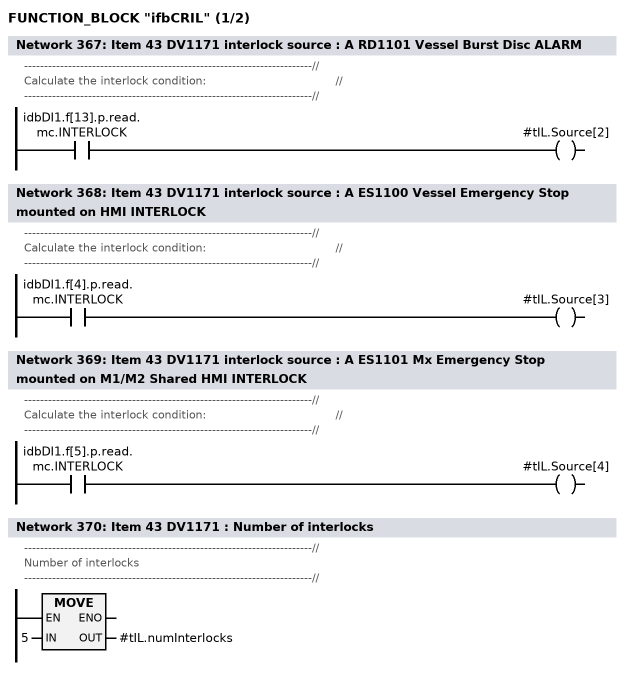
    A idbDI1.f[13].p.read.mc.INTERLOCK;
    = #tIL.Source[2];

NETWORK
TITLE = Item 43 DV1171 interlock source : A ES1100 Vessel Emergency Stop mounted on HMI INTERLOCK
    //------------------------------------------------------------------------//
    // Calculate the interlock condition:                                     //
    //------------------------------------------------------------------------//
    A idbDI1.f[4].p.read.mc.INTERLOCK;
    = #tIL.Source[3];

NETWORK
TITLE = Item 43 DV1171 interlock source : A ES1101 Mx Emergency Stop mounted on M1/M2 Shared HMI INTERLOCK
    //------------------------------------------------------------------------//
    // Calculate the interlock condition:                                     //
    //------------------------------------------------------------------------//
    A idbDI1.f[5].p.read.mc.INTERLOCK;
    = #tIL.Source[4];


NETWORK
TITLE = Item 43 DV1171 : Number of interlocks
    //------------------------------------------------------------------------//
    // Number of interlocks
    //------------------------------------------------------------------------//
    L 5;
    T #tIL.numInterlocks;

NETWORK
TITLE = Item 43 DV1171 : Aggregate individual interlocks into overall INTERLOCK flag
    //------------------------------------------------------------------------//
    // Determine if an interlock is raised:                                   //
    //------------------------------------------------------------------------//
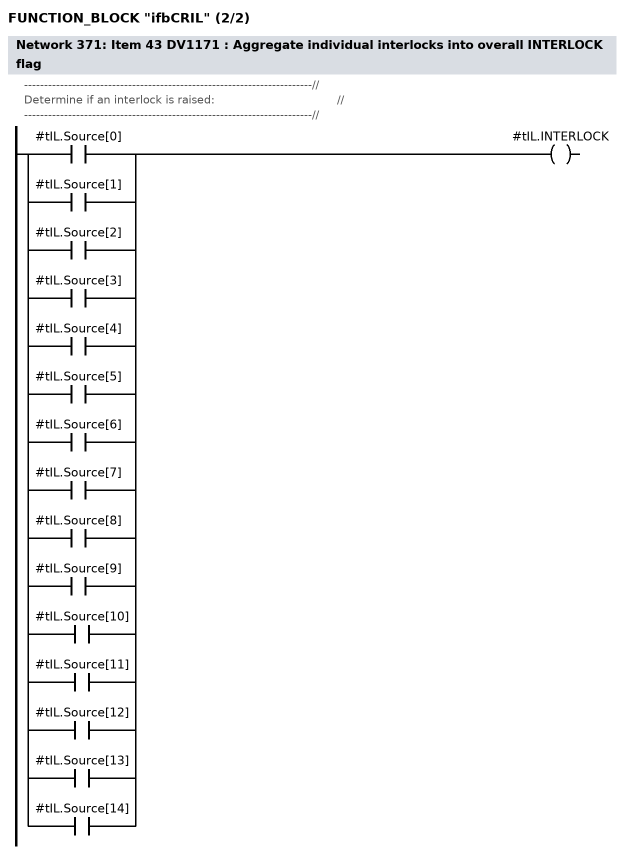
    O #tIL.Source[0];
    O #tIL.Source[1];
    O #tIL.Source[2];
    O #tIL.Source[3];
    O #tIL.Source[4];
    O #tIL.Source[5];
    O #tIL.Source[6];
    O #tIL.Source[7];
    O #tIL.Source[8];
    O #tIL.Source[9];
    O #tIL.Source[10];
    O #tIL.Source[11];
    O #tIL.Source[12];
    O #tIL.Source[13];
    O #tIL.Source[14];
    = #tIL.INTERLOCK;

NETWORK
TITLE = Item 43 DV1171 : Update the instance data
    //------------------------------------------------------------------------//
    // Update the instance DB with the calculated interlock flags:            //
    //------------------------------------------------------------------------//
    CALL MOVE
    {value_type := 'Variant'}
    (   IN                   := #tIL ,
        OUT                  := #p[43]
    );

NETWORK
TITLE = Item 44 DV1173 : MMFLx Inline Heat Exchanger inlet valve initialise variables
    //------------------------------------------------------------------------//
    // CRITICAL INTERLOCK   CRITICAL INTERLOCK   CRITICAL INTERLOCK   CRITICA //
    // CRITICAL INTERLOCK   CRITICAL INTERLOCK   CRITICAL INTERLOCK   CRITICA //
    //                                                                        //
    // Clear the interlock flag:                                              //
    //------------------------------------------------------------------------//
    A "alwaysLow";
    = #tIL.INTERLOCK;

    //------------------------------------------------------------------------//
    // Clear all interlock values to initialise them to off:                  //
    //------------------------------------------------------------------------//
    CALL FILL_BLK
    {value_type := 'Bool', count_type := 'UInt'}
    (   IN                   := 0 ,
        COUNT                := 15 ,
        OUT                  := #tIL.Source[0]
    );


NETWORK
TITLE = Item 44 DV1173 interlock source : AN ZSC1113 MMFLx Filtration Inlet Flowpath Indicator IN   AN ZSC1115 MMFLx Filtration Inlet CIP & SIP Flowpath Indicator IN
    //------------------------------------------------------------------------//
    // Calculate the interlock condition:                                     //
    //------------------------------------------------------------------------//
    AN(;
    L "idbZSC2".f[5].p.read.mc.STATE;
    L "dbCONST".BLK.ZSC2.STATE.IN;
    ==I;
    );
AN(;
    L "idbZSC2".f[6].p.read.mc.STATE;
    L "dbCONST".BLK.ZSC2.STATE.IN;
    ==I;
    );
    = #tIL.Source[0];

NETWORK
TITLE = Item 44 DV1173 interlock source : A RD1101 Vessel Burst Disc ALARM
    //------------------------------------------------------------------------//
    // Calculate the interlock condition:                                     //
    //------------------------------------------------------------------------//
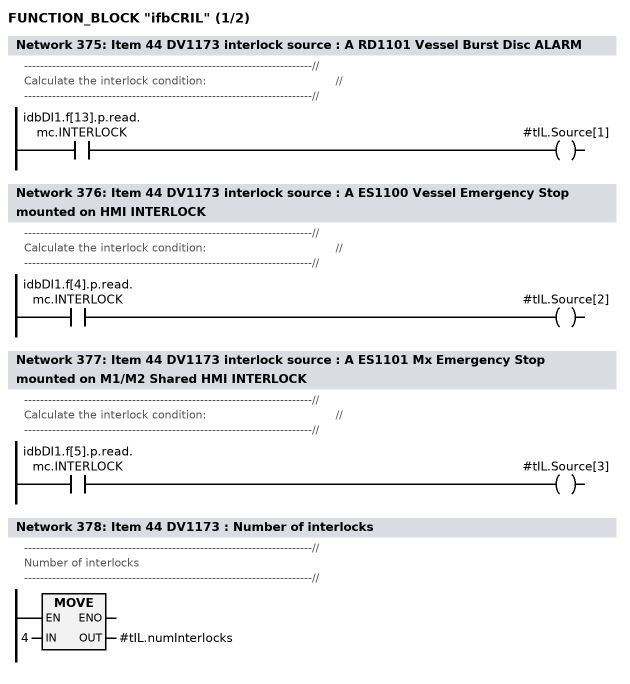
    A idbDI1.f[13].p.read.mc.INTERLOCK;
    = #tIL.Source[1];

NETWORK
TITLE = Item 44 DV1173 interlock source : A ES1100 Vessel Emergency Stop mounted on HMI INTERLOCK
    //------------------------------------------------------------------------//
    // Calculate the interlock condition:                                     //
    //------------------------------------------------------------------------//
    A idbDI1.f[4].p.read.mc.INTERLOCK;
    = #tIL.Source[2];

NETWORK
TITLE = Item 44 DV1173 interlock source : A ES1101 Mx Emergency Stop mounted on M1/M2 Shared HMI INTERLOCK
    //------------------------------------------------------------------------//
    // Calculate the interlock condition:                                     //
    //------------------------------------------------------------------------//
    A idbDI1.f[5].p.read.mc.INTERLOCK;
    = #tIL.Source[3];


NETWORK
TITLE = Item 44 DV1173 : Number of interlocks
    //------------------------------------------------------------------------//
    // Number of interlocks
    //------------------------------------------------------------------------//
    L 4;
    T #tIL.numInterlocks;

NETWORK
TITLE = Item 44 DV1173 : Aggregate individual interlocks into overall INTERLOCK flag
    //------------------------------------------------------------------------//
    // Determine if an interlock is raised:                                   //
    //------------------------------------------------------------------------//
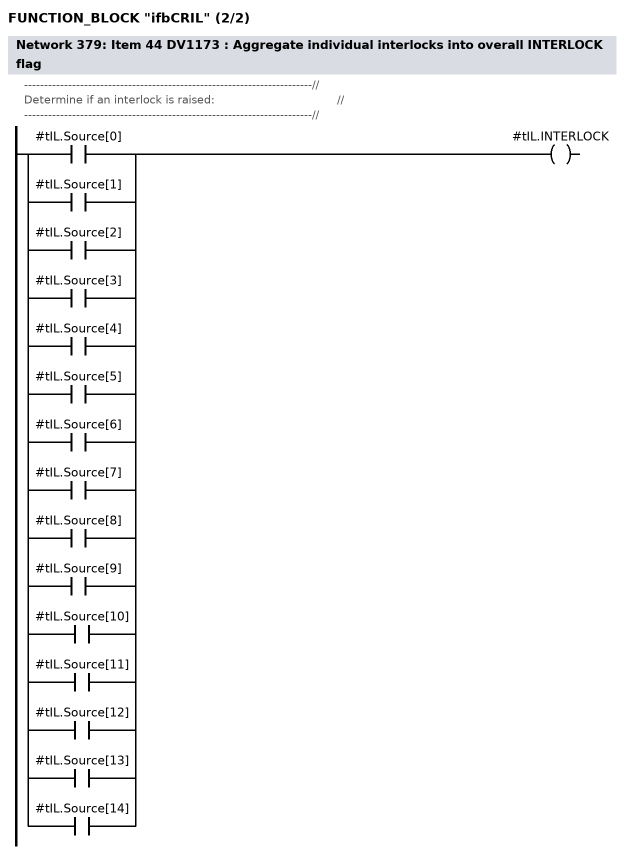
    O #tIL.Source[0];
    O #tIL.Source[1];
    O #tIL.Source[2];
    O #tIL.Source[3];
    O #tIL.Source[4];
    O #tIL.Source[5];
    O #tIL.Source[6];
    O #tIL.Source[7];
    O #tIL.Source[8];
    O #tIL.Source[9];
    O #tIL.Source[10];
    O #tIL.Source[11];
    O #tIL.Source[12];
    O #tIL.Source[13];
    O #tIL.Source[14];
    = #tIL.INTERLOCK;

NETWORK
TITLE = Item 44 DV1173 : Update the instance data
    //------------------------------------------------------------------------//
    // Update the instance DB with the calculated interlock flags:            //
    //------------------------------------------------------------------------//
    CALL MOVE
    {value_type := 'Variant'}
    (   IN                   := #tIL ,
        OUT                  := #p[44]
    );

NETWORK
TITLE = Item 45 DV2101 : Vent Valve initialise variables
    //------------------------------------------------------------------------//
    // CRITICAL INTERLOCK   CRITICAL INTERLOCK   CRITICAL INTERLOCK   CRITICA //
    // CRITICAL INTERLOCK   CRITICAL INTERLOCK   CRITICAL INTERLOCK   CRITICA //
    //                                                                        //
    // Clear the interlock flag:                                              //
    //------------------------------------------------------------------------//
    A "alwaysLow";
    = #tIL.INTERLOCK;

    //------------------------------------------------------------------------//
    // Clear all interlock values to initialise them to off:                  //
    //------------------------------------------------------------------------//
    CALL FILL_BLK
    {value_type := 'Bool', count_type := 'UInt'}
    (   IN                   := 0 ,
        COUNT                := 15 ,
        OUT                  := #tIL.Source[0]
    );


NETWORK
TITLE = Item 45 DV2101 interlock source : A RD2101 Vessel Burst Disc ALARM
    //------------------------------------------------------------------------//
    // Calculate the interlock condition:                                     //
    //------------------------------------------------------------------------//
    A idbDI1.f[14].p.read.mc.INTERLOCK;
    = #tIL.Source[0];

NETWORK
TITLE = Item 45 DV2101 interlock source : A ES2100 Vessel Emergency Stop mounted on HMI INTERLOCK
    //------------------------------------------------------------------------//
    // Calculate the interlock condition:                                     //
    //------------------------------------------------------------------------//
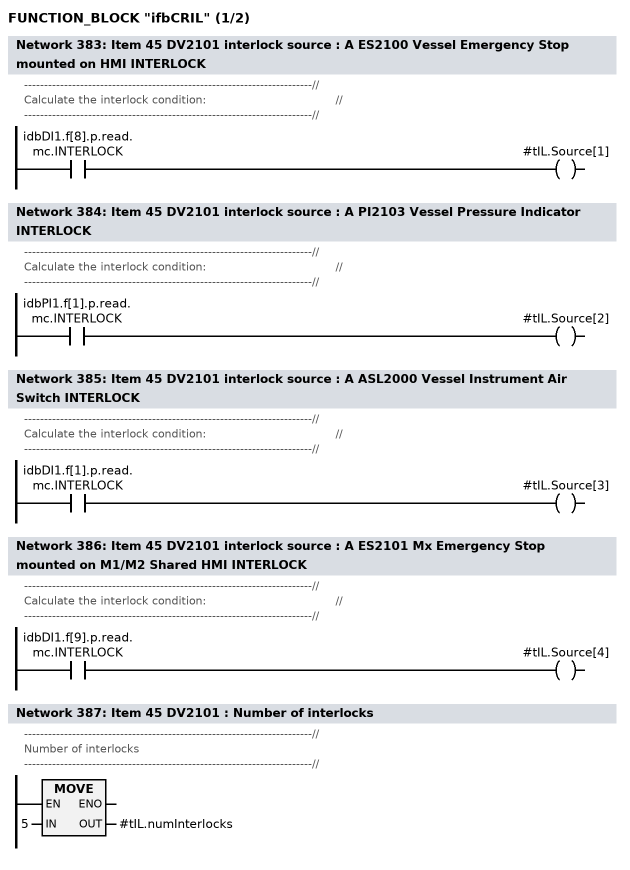
    A idbDI1.f[8].p.read.mc.INTERLOCK;
    = #tIL.Source[1];

NETWORK
TITLE = Item 45 DV2101 interlock source : A PI2103 Vessel Pressure Indicator INTERLOCK
    //------------------------------------------------------------------------//
    // Calculate the interlock condition:                                     //
    //------------------------------------------------------------------------//
    A idbPI1.f[1].p.read.mc.INTERLOCK;
    = #tIL.Source[2];

NETWORK
TITLE = Item 45 DV2101 interlock source : A ASL2000 Vessel Instrument Air Switch INTERLOCK
    //------------------------------------------------------------------------//
    // Calculate the interlock condition:                                     //
    //------------------------------------------------------------------------//
    A idbDI1.f[1].p.read.mc.INTERLOCK;
    = #tIL.Source[3];

NETWORK
TITLE = Item 45 DV2101 interlock source : A ES2101 Mx Emergency Stop mounted on M1/M2 Shared HMI INTERLOCK
    //------------------------------------------------------------------------//
    // Calculate the interlock condition:                                     //
    //------------------------------------------------------------------------//
    A idbDI1.f[9].p.read.mc.INTERLOCK;
    = #tIL.Source[4];


NETWORK
TITLE = Item 45 DV2101 : Number of interlocks
    //------------------------------------------------------------------------//
    // Number of interlocks
    //------------------------------------------------------------------------//
    L 5;
    T #tIL.numInterlocks;

NETWORK
TITLE = Item 45 DV2101 : Aggregate individual interlocks into overall INTERLOCK flag
    //------------------------------------------------------------------------//
    // Determine if an interlock is raised:                                   //
    //------------------------------------------------------------------------//
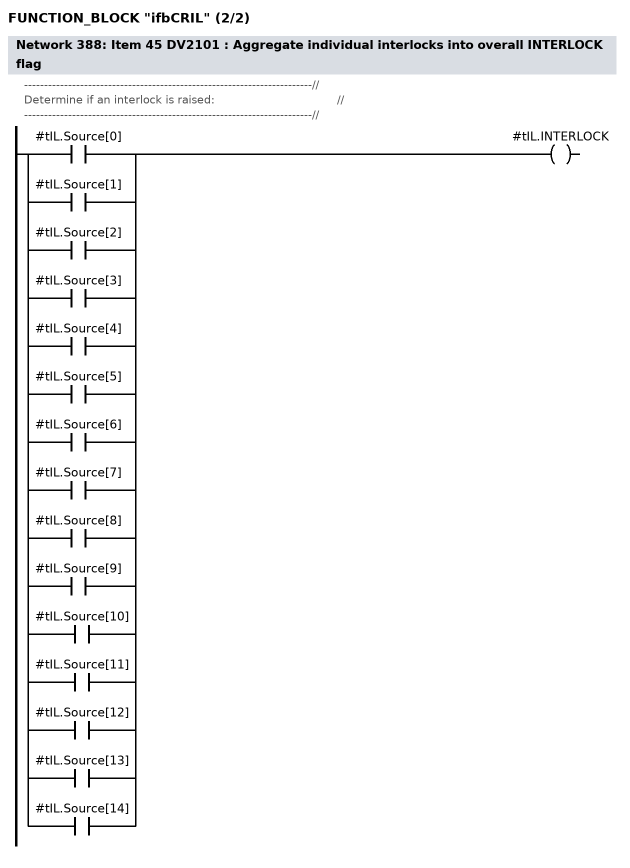
    O #tIL.Source[0];
    O #tIL.Source[1];
    O #tIL.Source[2];
    O #tIL.Source[3];
    O #tIL.Source[4];
    O #tIL.Source[5];
    O #tIL.Source[6];
    O #tIL.Source[7];
    O #tIL.Source[8];
    O #tIL.Source[9];
    O #tIL.Source[10];
    O #tIL.Source[11];
    O #tIL.Source[12];
    O #tIL.Source[13];
    O #tIL.Source[14];
    = #tIL.INTERLOCK;

NETWORK
TITLE = Item 45 DV2101 : Update the instance data
    //------------------------------------------------------------------------//
    // Update the instance DB with the calculated interlock flags:            //
    //------------------------------------------------------------------------//
    CALL MOVE
    {value_type := 'Variant'}
    (   IN                   := #tIL ,
        OUT                  := #p[45]
    );

NETWORK
TITLE = Item 46 DV2103 : HP CA Supply Valve initialise variables
    //------------------------------------------------------------------------//
    // CRITICAL INTERLOCK   CRITICAL INTERLOCK   CRITICAL INTERLOCK   CRITICA //
    // CRITICAL INTERLOCK   CRITICAL INTERLOCK   CRITICAL INTERLOCK   CRITICA //
    //                                                                        //
    // Clear the interlock flag:                                              //
    //------------------------------------------------------------------------//
    A "alwaysLow";
    = #tIL.INTERLOCK;

    //------------------------------------------------------------------------//
    // Clear all interlock values to initialise them to off:                  //
    //------------------------------------------------------------------------//
    CALL FILL_BLK
    {value_type := 'Bool', count_type := 'UInt'}
    (   IN                   := 0 ,
        COUNT                := 15 ,
        OUT                  := #tIL.Source[0]
    );


NETWORK
TITLE = Item 46 DV2103 interlock source : A RD2101 Vessel Burst Disc ALARM
    //------------------------------------------------------------------------//
    // Calculate the interlock condition:                                     //
    //------------------------------------------------------------------------//
    A idbDI1.f[14].p.read.mc.INTERLOCK;
    = #tIL.Source[0];

NETWORK
TITLE = Item 46 DV2103 interlock source : A ES2100 Vessel Emergency Stop mounted on HMI INTERLOCK
    //------------------------------------------------------------------------//
    // Calculate the interlock condition:                                     //
    //------------------------------------------------------------------------//
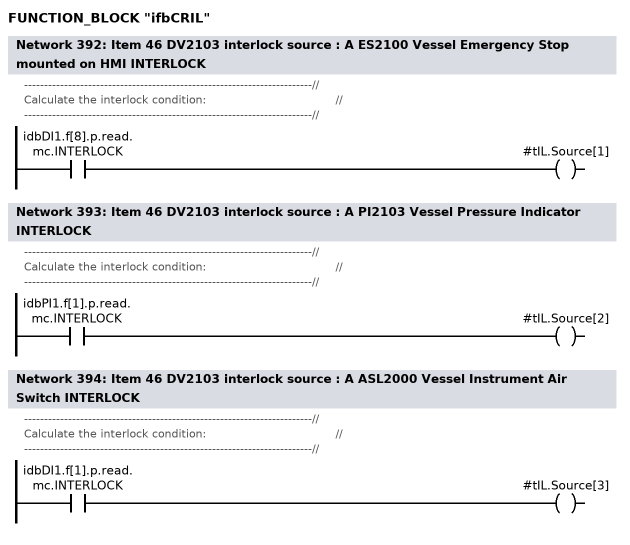
    A idbDI1.f[8].p.read.mc.INTERLOCK;
    = #tIL.Source[1];

NETWORK
TITLE = Item 46 DV2103 interlock source : A PI2103 Vessel Pressure Indicator INTERLOCK
    //------------------------------------------------------------------------//
    // Calculate the interlock condition:                                     //
    //------------------------------------------------------------------------//
    A idbPI1.f[1].p.read.mc.INTERLOCK;
    = #tIL.Source[2];

NETWORK
TITLE = Item 46 DV2103 interlock source : A ASL2000 Vessel Instrument Air Switch INTERLOCK
    //------------------------------------------------------------------------//
    // Calculate the interlock condition:                                     //
    //------------------------------------------------------------------------//
    A idbDI1.f[1].p.read.mc.INTERLOCK;
    = #tIL.Source[3];

NETWORK
TITLE = Item 46 DV2103 interlock source : AN ZSC2101 Vessel Manway Closed Indicator CLOSED
    //------------------------------------------------------------------------//
    // Calculate the interlock condition:                                     //
    //------------------------------------------------------------------------//
    AN(;
    L "idbZSC1".f[1].p.read.mc.STATE;
    L "dbCONST".BLK.ZSC1.STATE.CLOSED;
    ==I;
    );
    = #tIL.Source[4];

NETWORK
TITLE = Item 46 DV2103 interlock source : A ES2101 Mx Emergency Stop mounted on M1/M2 Shared HMI INTERLOCK
    //------------------------------------------------------------------------//
    // Calculate the interlock condition:                                     //
    //------------------------------------------------------------------------//
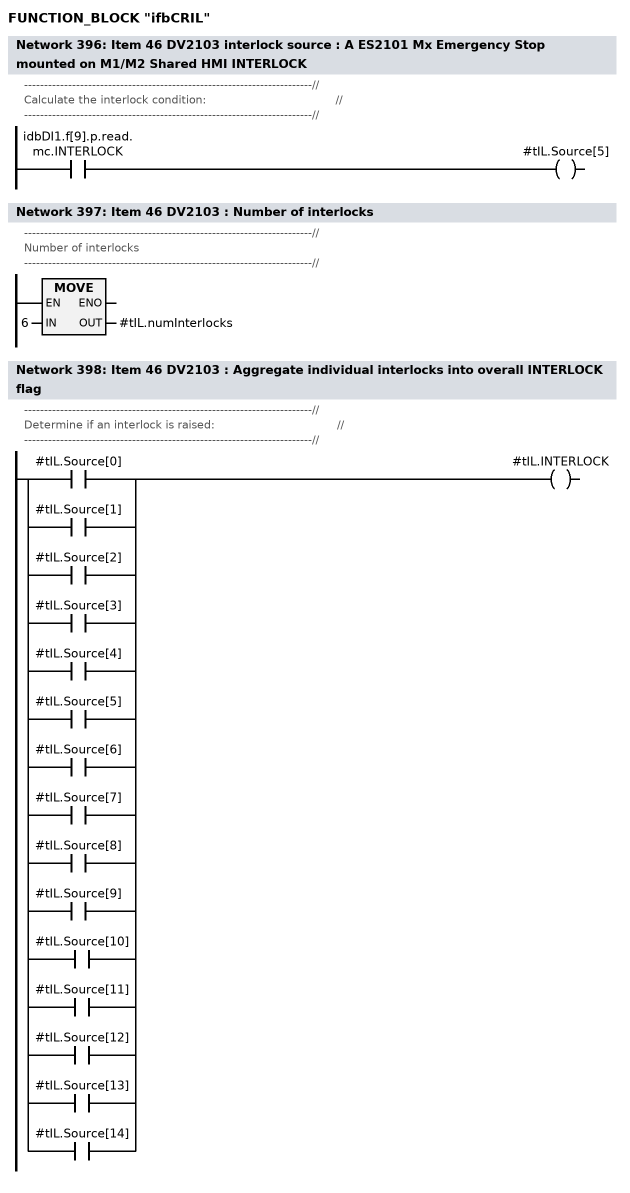
    A idbDI1.f[9].p.read.mc.INTERLOCK;
    = #tIL.Source[5];


NETWORK
TITLE = Item 46 DV2103 : Number of interlocks
    //------------------------------------------------------------------------//
    // Number of interlocks
    //------------------------------------------------------------------------//
    L 6;
    T #tIL.numInterlocks;

NETWORK
TITLE = Item 46 DV2103 : Aggregate individual interlocks into overall INTERLOCK flag
    //------------------------------------------------------------------------//
    // Determine if an interlock is raised:                                   //
    //------------------------------------------------------------------------//
    O #tIL.Source[0];
    O #tIL.Source[1];
    O #tIL.Source[2];
    O #tIL.Source[3];
    O #tIL.Source[4];
    O #tIL.Source[5];
    O #tIL.Source[6];
    O #tIL.Source[7];
    O #tIL.Source[8];
    O #tIL.Source[9];
    O #tIL.Source[10];
    O #tIL.Source[11];
    O #tIL.Source[12];
    O #tIL.Source[13];
    O #tIL.Source[14];
    = #tIL.INTERLOCK;

NETWORK
TITLE = Item 46 DV2103 : Update the instance data
    //------------------------------------------------------------------------//
    // Update the instance DB with the calculated interlock flags:            //
    //------------------------------------------------------------------------//
    CALL MOVE
    {value_type := 'Variant'}
    (   IN                   := #tIL ,
        OUT                  := #p[46]
    );

NETWORK
TITLE = Item 47 DV2105 : LP CA Supply Valve initialise variables
    //------------------------------------------------------------------------//
    // CRITICAL INTERLOCK   CRITICAL INTERLOCK   CRITICAL INTERLOCK   CRITICA //
    // CRITICAL INTERLOCK   CRITICAL INTERLOCK   CRITICAL INTERLOCK   CRITICA //
    //                                                                        //
    // Clear the interlock flag:                                              //
    //------------------------------------------------------------------------//
    A "alwaysLow";
    = #tIL.INTERLOCK;

    //------------------------------------------------------------------------//
    // Clear all interlock values to initialise them to off:                  //
    //------------------------------------------------------------------------//
    CALL FILL_BLK
    {value_type := 'Bool', count_type := 'UInt'}
    (   IN                   := 0 ,
        COUNT                := 15 ,
        OUT                  := #tIL.Source[0]
    );


NETWORK
TITLE = Item 47 DV2105 interlock source : A RD2101 Vessel Burst Disc ALARM
    //------------------------------------------------------------------------//
    // Calculate the interlock condition:                                     //
    //------------------------------------------------------------------------//
    A idbDI1.f[14].p.read.mc.INTERLOCK;
    = #tIL.Source[0];

NETWORK
TITLE = Item 47 DV2105 interlock source : A ES2100 Vessel Emergency Stop mounted on HMI INTERLOCK
    //------------------------------------------------------------------------//
    // Calculate the interlock condition:                                     //
    //------------------------------------------------------------------------//
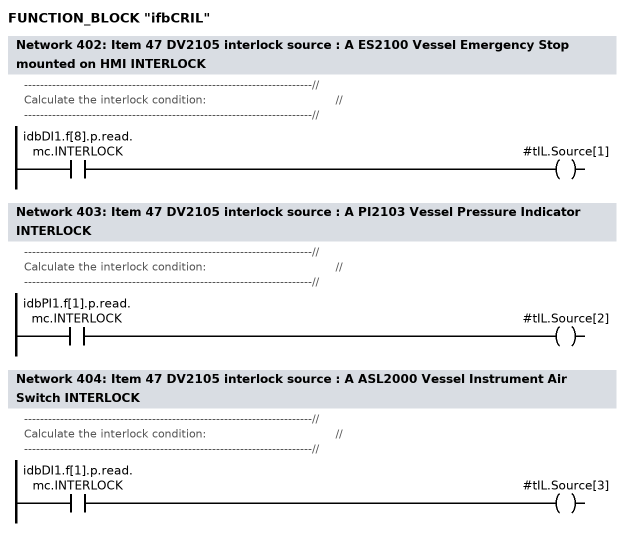
    A idbDI1.f[8].p.read.mc.INTERLOCK;
    = #tIL.Source[1];

NETWORK
TITLE = Item 47 DV2105 interlock source : A PI2103 Vessel Pressure Indicator INTERLOCK
    //------------------------------------------------------------------------//
    // Calculate the interlock condition:                                     //
    //------------------------------------------------------------------------//
    A idbPI1.f[1].p.read.mc.INTERLOCK;
    = #tIL.Source[2];

NETWORK
TITLE = Item 47 DV2105 interlock source : A ASL2000 Vessel Instrument Air Switch INTERLOCK
    //------------------------------------------------------------------------//
    // Calculate the interlock condition:                                     //
    //------------------------------------------------------------------------//
    A idbDI1.f[1].p.read.mc.INTERLOCK;
    = #tIL.Source[3];

NETWORK
TITLE = Item 47 DV2105 interlock source : AN ZSC2101 Vessel Manway Closed Indicator CLOSED
    //------------------------------------------------------------------------//
    // Calculate the interlock condition:                                     //
    //------------------------------------------------------------------------//
    AN(;
    L "idbZSC1".f[1].p.read.mc.STATE;
    L "dbCONST".BLK.ZSC1.STATE.CLOSED;
    ==I;
    );
    = #tIL.Source[4];

NETWORK
TITLE = Item 47 DV2105 interlock source : A ES2101 Mx Emergency Stop mounted on M1/M2 Shared HMI INTERLOCK
    //------------------------------------------------------------------------//
    // Calculate the interlock condition:                                     //
    //------------------------------------------------------------------------//
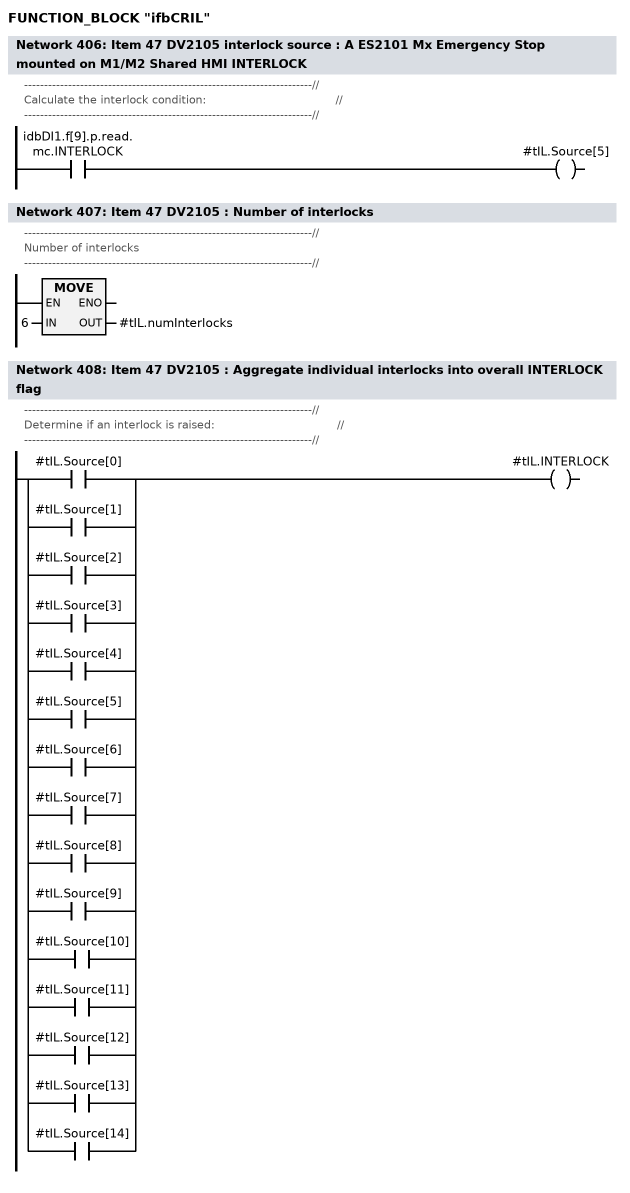
    A idbDI1.f[9].p.read.mc.INTERLOCK;
    = #tIL.Source[5];


NETWORK
TITLE = Item 47 DV2105 : Number of interlocks
    //------------------------------------------------------------------------//
    // Number of interlocks
    //------------------------------------------------------------------------//
    L 6;
    T #tIL.numInterlocks;

NETWORK
TITLE = Item 47 DV2105 : Aggregate individual interlocks into overall INTERLOCK flag
    //------------------------------------------------------------------------//
    // Determine if an interlock is raised:                                   //
    //------------------------------------------------------------------------//
    O #tIL.Source[0];
    O #tIL.Source[1];
    O #tIL.Source[2];
    O #tIL.Source[3];
    O #tIL.Source[4];
    O #tIL.Source[5];
    O #tIL.Source[6];
    O #tIL.Source[7];
    O #tIL.Source[8];
    O #tIL.Source[9];
    O #tIL.Source[10];
    O #tIL.Source[11];
    O #tIL.Source[12];
    O #tIL.Source[13];
    O #tIL.Source[14];
    = #tIL.INTERLOCK;

NETWORK
TITLE = Item 47 DV2105 : Update the instance data
    //------------------------------------------------------------------------//
    // Update the instance DB with the calculated interlock flags:            //
    //------------------------------------------------------------------------//
    CALL MOVE
    {value_type := 'Variant'}
    (   IN                   := #tIL ,
        OUT                  := #p[47]
    );

NETWORK
TITLE = Item 48 DV2107 : Vacuum valve initialise variables
    //------------------------------------------------------------------------//
    // CRITICAL INTERLOCK   CRITICAL INTERLOCK   CRITICAL INTERLOCK   CRITICA //
    // CRITICAL INTERLOCK   CRITICAL INTERLOCK   CRITICAL INTERLOCK   CRITICA //
    //                                                                        //
    // Clear the interlock flag:                                              //
    //------------------------------------------------------------------------//
    A "alwaysLow";
    = #tIL.INTERLOCK;

    //------------------------------------------------------------------------//
    // Clear all interlock values to initialise them to off:                  //
    //------------------------------------------------------------------------//
    CALL FILL_BLK
    {value_type := 'Bool', count_type := 'UInt'}
    (   IN                   := 0 ,
        COUNT                := 15 ,
        OUT                  := #tIL.Source[0]
    );


NETWORK
TITLE = Item 48 DV2107 interlock source : A RD2101 Vessel Burst Disc ALARM
    //------------------------------------------------------------------------//
    // Calculate the interlock condition:                                     //
    //------------------------------------------------------------------------//
    A idbDI1.f[14].p.read.mc.INTERLOCK;
    = #tIL.Source[0];

NETWORK
TITLE = Item 48 DV2107 interlock source : A ES2100 Vessel Emergency Stop mounted on HMI INTERLOCK
    //------------------------------------------------------------------------//
    // Calculate the interlock condition:                                     //
    //------------------------------------------------------------------------//
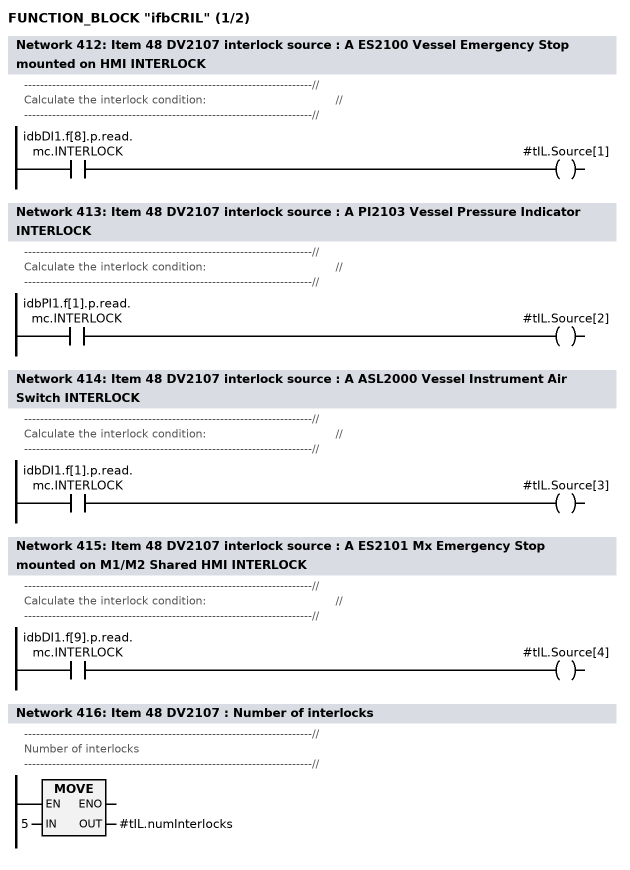
    A idbDI1.f[8].p.read.mc.INTERLOCK;
    = #tIL.Source[1];

NETWORK
TITLE = Item 48 DV2107 interlock source : A PI2103 Vessel Pressure Indicator INTERLOCK
    //------------------------------------------------------------------------//
    // Calculate the interlock condition:                                     //
    //------------------------------------------------------------------------//
    A idbPI1.f[1].p.read.mc.INTERLOCK;
    = #tIL.Source[2];

NETWORK
TITLE = Item 48 DV2107 interlock source : A ASL2000 Vessel Instrument Air Switch INTERLOCK
    //------------------------------------------------------------------------//
    // Calculate the interlock condition:                                     //
    //------------------------------------------------------------------------//
    A idbDI1.f[1].p.read.mc.INTERLOCK;
    = #tIL.Source[3];

NETWORK
TITLE = Item 48 DV2107 interlock source : A ES2101 Mx Emergency Stop mounted on M1/M2 Shared HMI INTERLOCK
    //------------------------------------------------------------------------//
    // Calculate the interlock condition:                                     //
    //------------------------------------------------------------------------//
    A idbDI1.f[9].p.read.mc.INTERLOCK;
    = #tIL.Source[4];


NETWORK
TITLE = Item 48 DV2107 : Number of interlocks
    //------------------------------------------------------------------------//
    // Number of interlocks
    //------------------------------------------------------------------------//
    L 5;
    T #tIL.numInterlocks;

NETWORK
TITLE = Item 48 DV2107 : Aggregate individual interlocks into overall INTERLOCK flag
    //------------------------------------------------------------------------//
    // Determine if an interlock is raised:                                   //
    //------------------------------------------------------------------------//
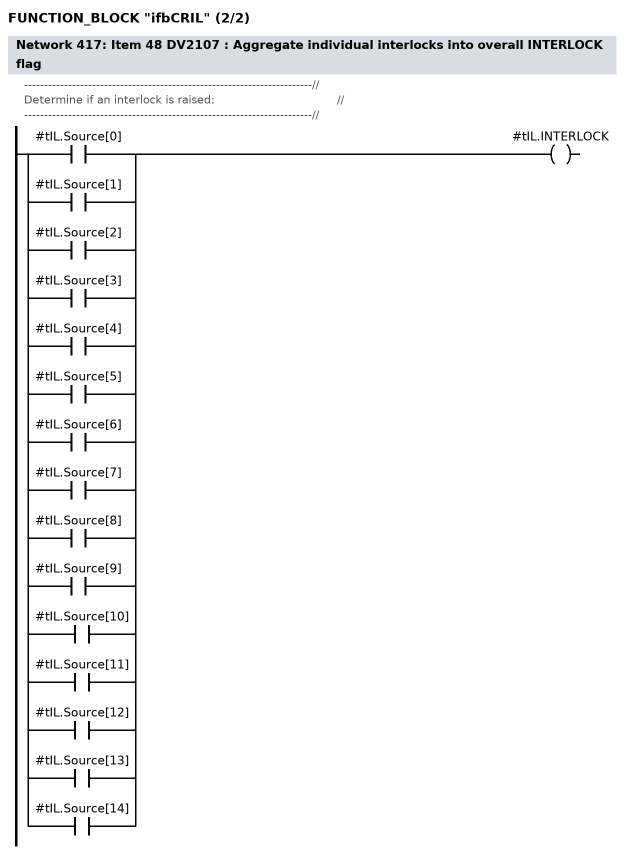
    O #tIL.Source[0];
    O #tIL.Source[1];
    O #tIL.Source[2];
    O #tIL.Source[3];
    O #tIL.Source[4];
    O #tIL.Source[5];
    O #tIL.Source[6];
    O #tIL.Source[7];
    O #tIL.Source[8];
    O #tIL.Source[9];
    O #tIL.Source[10];
    O #tIL.Source[11];
    O #tIL.Source[12];
    O #tIL.Source[13];
    O #tIL.Source[14];
    = #tIL.INTERLOCK;

NETWORK
TITLE = Item 48 DV2107 : Update the instance data
    //------------------------------------------------------------------------//
    // Update the instance DB with the calculated interlock flags:            //
    //------------------------------------------------------------------------//
    CALL MOVE
    {value_type := 'Variant'}
    (   IN                   := #tIL ,
        OUT                  := #p[48]
    );

NETWORK
TITLE = Item 49 DV2109 : PS Supply for WFI Loop initialise variables
    //------------------------------------------------------------------------//
    // CRITICAL INTERLOCK   CRITICAL INTERLOCK   CRITICAL INTERLOCK   CRITICA //
    // CRITICAL INTERLOCK   CRITICAL INTERLOCK   CRITICAL INTERLOCK   CRITICA //
    //                                                                        //
    // Clear the interlock flag:                                              //
    //------------------------------------------------------------------------//
    A "alwaysLow";
    = #tIL.INTERLOCK;

    //------------------------------------------------------------------------//
    // Clear all interlock values to initialise them to off:                  //
    //------------------------------------------------------------------------//
    CALL FILL_BLK
    {value_type := 'Bool', count_type := 'UInt'}
    (   IN                   := 0 ,
        COUNT                := 15 ,
        OUT                  := #tIL.Source[0]
    );


NETWORK
TITLE = Item 49 DV2109 interlock source : ON ZSC2107 Vessel inlet line Flowpath Indicator IN   ON ZSC2103 Vessel WFI Supply Flowpath Indicator IN
    //------------------------------------------------------------------------//
    // Calculate the interlock condition:                                     //
    //------------------------------------------------------------------------//
    ON(;
    L "idbZSC2".f[9].p.read.mc.STATE;
    L "dbCONST".BLK.ZSC2.STATE.IN;
    ==I;
    );
ON(;
    L "idbZSC2".f[7].p.read.mc.STATE;
    L "dbCONST".BLK.ZSC2.STATE.IN;
    ==I;
    );
    = #tIL.Source[0];

NETWORK
TITLE = Item 49 DV2109 interlock source : A DV2111 Vessel WFI Supply Valve OPENED
    //------------------------------------------------------------------------//
    // Calculate the interlock condition:                                     //
    //------------------------------------------------------------------------//
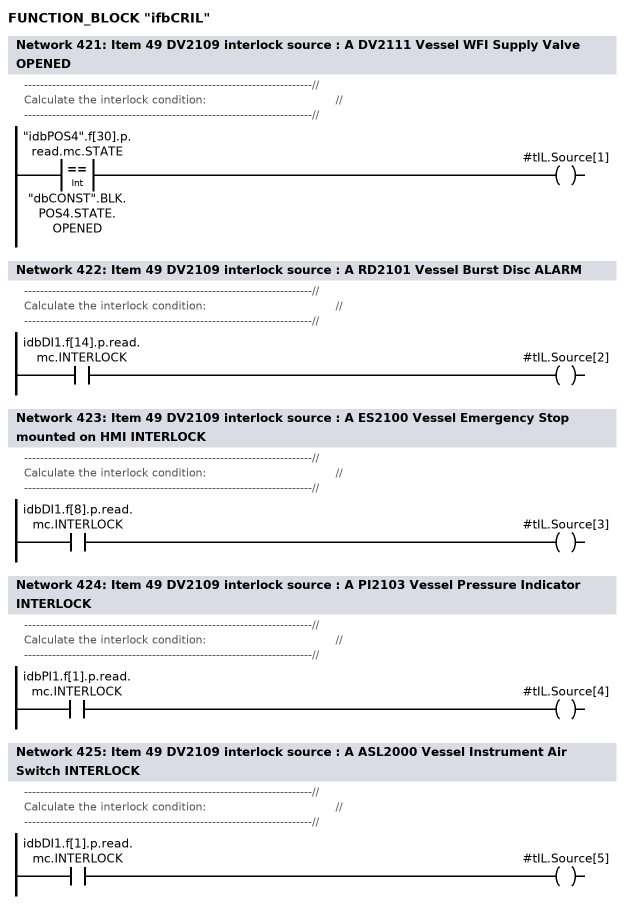
    A(;
    L "idbPOS4".f[30].p.read.mc.STATE;
    L "dbCONST".BLK.POS4.STATE.OPENED;
    ==I;
    );
    = #tIL.Source[1];

NETWORK
TITLE = Item 49 DV2109 interlock source : A RD2101 Vessel Burst Disc ALARM
    //------------------------------------------------------------------------//
    // Calculate the interlock condition:                                     //
    //------------------------------------------------------------------------//
    A idbDI1.f[14].p.read.mc.INTERLOCK;
    = #tIL.Source[2];

NETWORK
TITLE = Item 49 DV2109 interlock source : A ES2100 Vessel Emergency Stop mounted on HMI INTERLOCK
    //------------------------------------------------------------------------//
    // Calculate the interlock condition:                                     //
    //------------------------------------------------------------------------//
    A idbDI1.f[8].p.read.mc.INTERLOCK;
    = #tIL.Source[3];

NETWORK
TITLE = Item 49 DV2109 interlock source : A PI2103 Vessel Pressure Indicator INTERLOCK
    //------------------------------------------------------------------------//
    // Calculate the interlock condition:                                     //
    //------------------------------------------------------------------------//
    A idbPI1.f[1].p.read.mc.INTERLOCK;
    = #tIL.Source[4];

NETWORK
TITLE = Item 49 DV2109 interlock source : A ASL2000 Vessel Instrument Air Switch INTERLOCK
    //------------------------------------------------------------------------//
    // Calculate the interlock condition:                                     //
    //------------------------------------------------------------------------//
    A idbDI1.f[1].p.read.mc.INTERLOCK;
    = #tIL.Source[5];

NETWORK
TITLE = Item 49 DV2109 interlock source : AN ZSC2101 Vessel Manway Closed Indicator CLOSED
    //------------------------------------------------------------------------//
    // Calculate the interlock condition:                                     //
    //------------------------------------------------------------------------//
    AN(;
    L "idbZSC1".f[1].p.read.mc.STATE;
    L "dbCONST".BLK.ZSC1.STATE.CLOSED;
    ==I;
    );
    = #tIL.Source[6];

NETWORK
TITLE = Item 49 DV2109 interlock source : O MI2101 Mx Mass Indicator High High Alarm ALARM_HH   ON MI2101 Mx Mass Indicator Bad DQ DQ
    //------------------------------------------------------------------------//
    // Calculate the interlock condition:                                     //
    //------------------------------------------------------------------------//
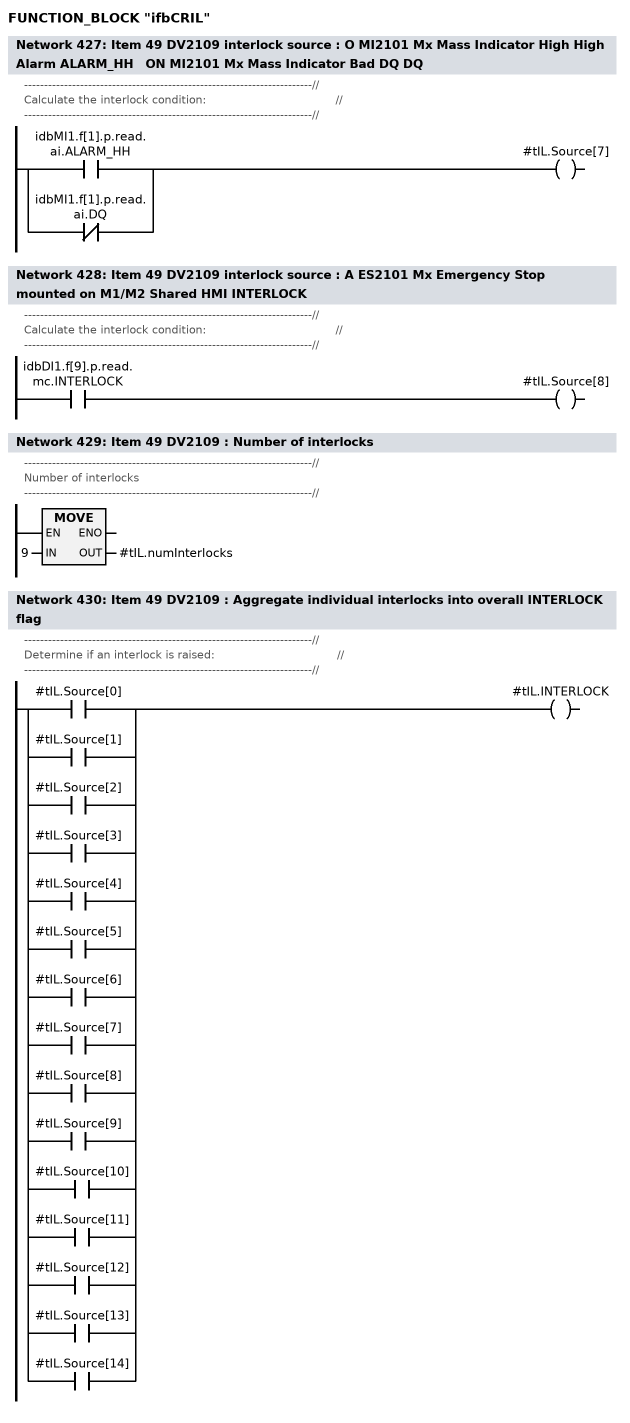
    O idbMI1.f[1].p.read.ai.ALARM_HH;
ON idbMI1.f[1].p.read.ai.DQ;
    = #tIL.Source[7];

NETWORK
TITLE = Item 49 DV2109 interlock source : A ES2101 Mx Emergency Stop mounted on M1/M2 Shared HMI INTERLOCK
    //------------------------------------------------------------------------//
    // Calculate the interlock condition:                                     //
    //------------------------------------------------------------------------//
    A idbDI1.f[9].p.read.mc.INTERLOCK;
    = #tIL.Source[8];


NETWORK
TITLE = Item 49 DV2109 : Number of interlocks
    //------------------------------------------------------------------------//
    // Number of interlocks
    //------------------------------------------------------------------------//
    L 9;
    T #tIL.numInterlocks;

NETWORK
TITLE = Item 49 DV2109 : Aggregate individual interlocks into overall INTERLOCK flag
    //------------------------------------------------------------------------//
    // Determine if an interlock is raised:                                   //
    //------------------------------------------------------------------------//
    O #tIL.Source[0];
    O #tIL.Source[1];
    O #tIL.Source[2];
    O #tIL.Source[3];
    O #tIL.Source[4];
    O #tIL.Source[5];
    O #tIL.Source[6];
    O #tIL.Source[7];
    O #tIL.Source[8];
    O #tIL.Source[9];
    O #tIL.Source[10];
    O #tIL.Source[11];
    O #tIL.Source[12];
    O #tIL.Source[13];
    O #tIL.Source[14];
    = #tIL.INTERLOCK;

NETWORK
TITLE = Item 49 DV2109 : Update the instance data
    //------------------------------------------------------------------------//
    // Update the instance DB with the calculated interlock flags:            //
    //------------------------------------------------------------------------//
    CALL MOVE
    {value_type := 'Variant'}
    (   IN                   := #tIL ,
        OUT                  := #p[49]
    );

NETWORK
TITLE = Item 50 DV2111 : WFI Supply Valve initialise variables
    //------------------------------------------------------------------------//
    // CRITICAL INTERLOCK   CRITICAL INTERLOCK   CRITICAL INTERLOCK   CRITICA //
    // CRITICAL INTERLOCK   CRITICAL INTERLOCK   CRITICAL INTERLOCK   CRITICA //
    //                                                                        //
    // Clear the interlock flag:                                              //
    //------------------------------------------------------------------------//
    A "alwaysLow";
    = #tIL.INTERLOCK;

    //------------------------------------------------------------------------//
    // Clear all interlock values to initialise them to off:                  //
    //------------------------------------------------------------------------//
    CALL FILL_BLK
    {value_type := 'Bool', count_type := 'UInt'}
    (   IN                   := 0 ,
        COUNT                := 15 ,
        OUT                  := #tIL.Source[0]
    );


NETWORK
TITLE = Item 50 DV2111 interlock source : ON ZSC2107 Vessel inlet line Flowpath Indicator IN   ON ZSC2103 Vessel WFI Supply Flowpath Indicator IN
    //------------------------------------------------------------------------//
    // Calculate the interlock condition:                                     //
    //------------------------------------------------------------------------//
    ON(;
    L "idbZSC2".f[9].p.read.mc.STATE;
    L "dbCONST".BLK.ZSC2.STATE.IN;
    ==I;
    );
ON(;
    L "idbZSC2".f[7].p.read.mc.STATE;
    L "dbCONST".BLK.ZSC2.STATE.IN;
    ==I;
    );
    = #tIL.Source[0];

NETWORK
TITLE = Item 50 DV2111 interlock source : A DV2109 Vessel PS Supply for WFI Loop OPENED
    //------------------------------------------------------------------------//
    // Calculate the interlock condition:                                     //
    //------------------------------------------------------------------------//
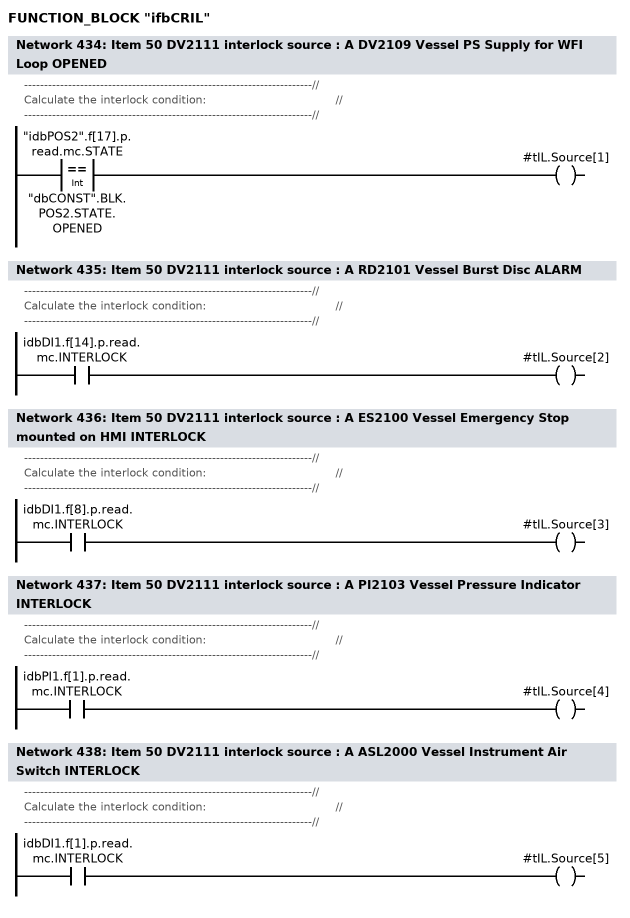
    A(;
    L "idbPOS2".f[17].p.read.mc.STATE;
    L "dbCONST".BLK.POS2.STATE.OPENED;
    ==I;
    );
    = #tIL.Source[1];

NETWORK
TITLE = Item 50 DV2111 interlock source : A RD2101 Vessel Burst Disc ALARM
    //------------------------------------------------------------------------//
    // Calculate the interlock condition:                                     //
    //------------------------------------------------------------------------//
    A idbDI1.f[14].p.read.mc.INTERLOCK;
    = #tIL.Source[2];

NETWORK
TITLE = Item 50 DV2111 interlock source : A ES2100 Vessel Emergency Stop mounted on HMI INTERLOCK
    //------------------------------------------------------------------------//
    // Calculate the interlock condition:                                     //
    //------------------------------------------------------------------------//
    A idbDI1.f[8].p.read.mc.INTERLOCK;
    = #tIL.Source[3];

NETWORK
TITLE = Item 50 DV2111 interlock source : A PI2103 Vessel Pressure Indicator INTERLOCK
    //------------------------------------------------------------------------//
    // Calculate the interlock condition:                                     //
    //------------------------------------------------------------------------//
    A idbPI1.f[1].p.read.mc.INTERLOCK;
    = #tIL.Source[4];

NETWORK
TITLE = Item 50 DV2111 interlock source : A ASL2000 Vessel Instrument Air Switch INTERLOCK
    //------------------------------------------------------------------------//
    // Calculate the interlock condition:                                     //
    //------------------------------------------------------------------------//
    A idbDI1.f[1].p.read.mc.INTERLOCK;
    = #tIL.Source[5];

NETWORK
TITLE = Item 50 DV2111 interlock source : AN ZSC2101 Vessel Manway Closed Indicator CLOSED
    //------------------------------------------------------------------------//
    // Calculate the interlock condition:                                     //
    //------------------------------------------------------------------------//
    AN(;
    L "idbZSC1".f[1].p.read.mc.STATE;
    L "dbCONST".BLK.ZSC1.STATE.CLOSED;
    ==I;
    );
    = #tIL.Source[6];

NETWORK
TITLE = Item 50 DV2111 interlock source : O MI2101 Mx Mass Indicator High High Alarm ALARM_HH   ON MI2101 Mx Mass Indicator Bad DQ DQ
    //------------------------------------------------------------------------//
    // Calculate the interlock condition:                                     //
    //------------------------------------------------------------------------//
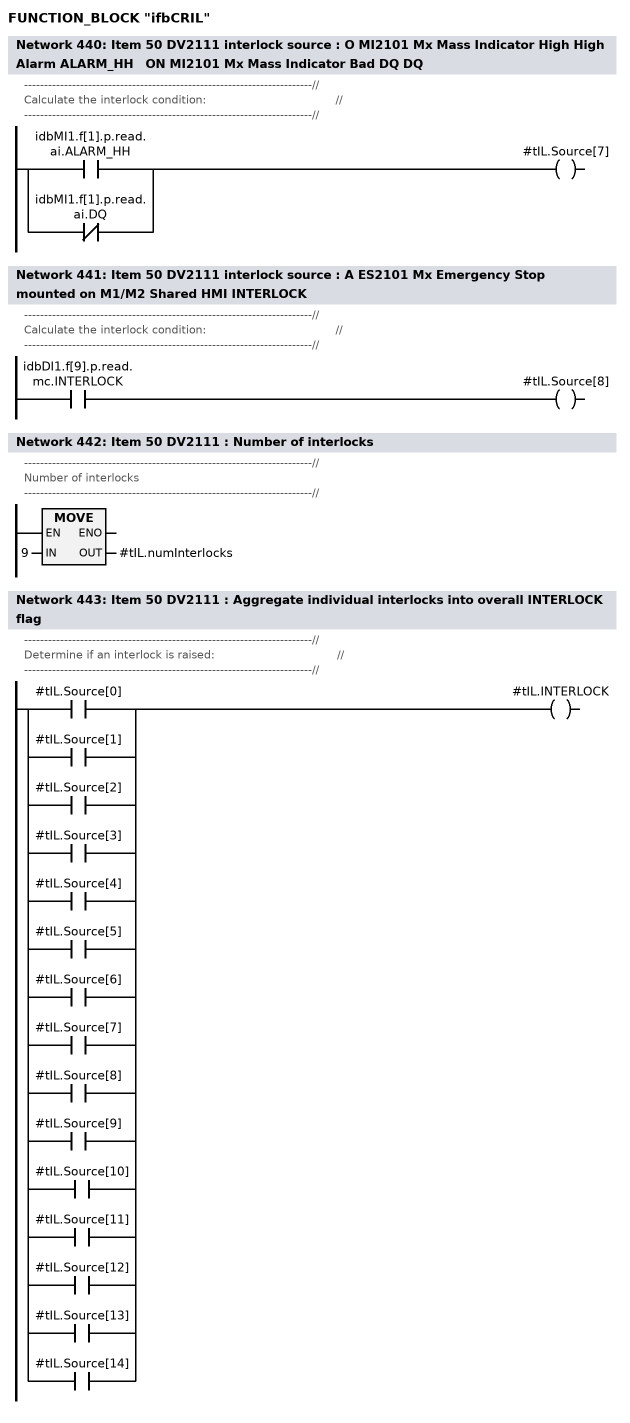
    O idbMI1.f[1].p.read.ai.ALARM_HH;
ON idbMI1.f[1].p.read.ai.DQ;
    = #tIL.Source[7];

NETWORK
TITLE = Item 50 DV2111 interlock source : A ES2101 Mx Emergency Stop mounted on M1/M2 Shared HMI INTERLOCK
    //------------------------------------------------------------------------//
    // Calculate the interlock condition:                                     //
    //------------------------------------------------------------------------//
    A idbDI1.f[9].p.read.mc.INTERLOCK;
    = #tIL.Source[8];


NETWORK
TITLE = Item 50 DV2111 : Number of interlocks
    //------------------------------------------------------------------------//
    // Number of interlocks
    //------------------------------------------------------------------------//
    L 9;
    T #tIL.numInterlocks;

NETWORK
TITLE = Item 50 DV2111 : Aggregate individual interlocks into overall INTERLOCK flag
    //------------------------------------------------------------------------//
    // Determine if an interlock is raised:                                   //
    //------------------------------------------------------------------------//
    O #tIL.Source[0];
    O #tIL.Source[1];
    O #tIL.Source[2];
    O #tIL.Source[3];
    O #tIL.Source[4];
    O #tIL.Source[5];
    O #tIL.Source[6];
    O #tIL.Source[7];
    O #tIL.Source[8];
    O #tIL.Source[9];
    O #tIL.Source[10];
    O #tIL.Source[11];
    O #tIL.Source[12];
    O #tIL.Source[13];
    O #tIL.Source[14];
    = #tIL.INTERLOCK;

NETWORK
TITLE = Item 50 DV2111 : Update the instance data
    //------------------------------------------------------------------------//
    // Update the instance DB with the calculated interlock flags:            //
    //------------------------------------------------------------------------//
    CALL MOVE
    {value_type := 'Variant'}
    (   IN                   := #tIL ,
        OUT                  := #p[50]
    );

NETWORK
TITLE = Item 51 DV2113 : PW Supply Valve initialise variables
    //------------------------------------------------------------------------//
    // CRITICAL INTERLOCK   CRITICAL INTERLOCK   CRITICAL INTERLOCK   CRITICA //
    // CRITICAL INTERLOCK   CRITICAL INTERLOCK   CRITICAL INTERLOCK   CRITICA //
    //                                                                        //
    // Clear the interlock flag:                                              //
    //------------------------------------------------------------------------//
    A "alwaysLow";
    = #tIL.INTERLOCK;

    //------------------------------------------------------------------------//
    // Clear all interlock values to initialise them to off:                  //
    //------------------------------------------------------------------------//
    CALL FILL_BLK
    {value_type := 'Bool', count_type := 'UInt'}
    (   IN                   := 0 ,
        COUNT                := 15 ,
        OUT                  := #tIL.Source[0]
    );


NETWORK
TITLE = Item 51 DV2113 interlock source : ON ZSC2107 Vessel inlet line Flowpath Indicator IN   ON ZSC2105 Vessel PW Supply Flowpath Indicator IN
    //------------------------------------------------------------------------//
    // Calculate the interlock condition:                                     //
    //------------------------------------------------------------------------//
    ON(;
    L "idbZSC2".f[9].p.read.mc.STATE;
    L "dbCONST".BLK.ZSC2.STATE.IN;
    ==I;
    );
ON(;
    L "idbZSC2".f[8].p.read.mc.STATE;
    L "dbCONST".BLK.ZSC2.STATE.IN;
    ==I;
    );
    = #tIL.Source[0];

NETWORK
TITLE = Item 51 DV2113 interlock source : A DV2115 Vessel PS Supply for PW Loop OPENED
    //------------------------------------------------------------------------//
    // Calculate the interlock condition:                                     //
    //------------------------------------------------------------------------//
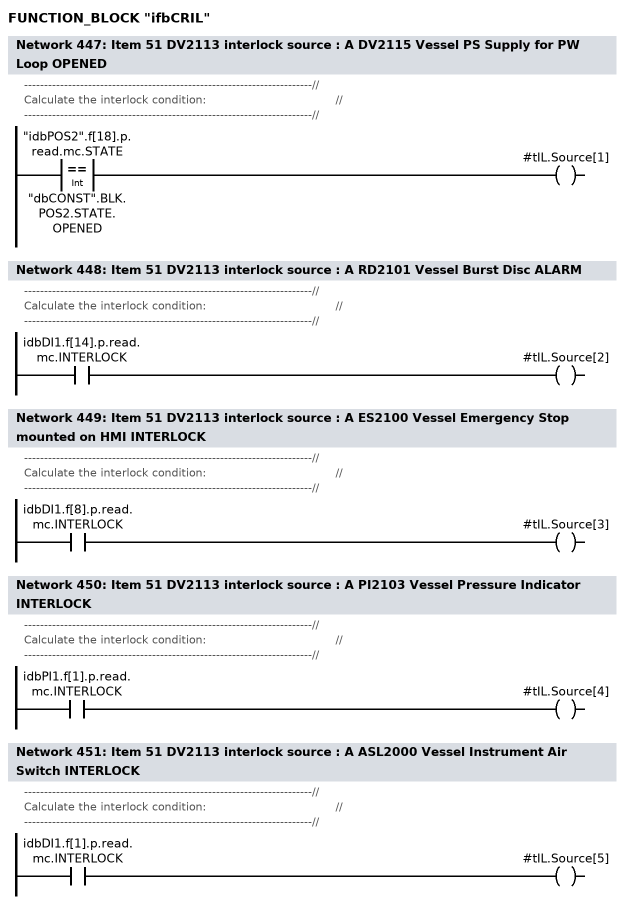
    A(;
    L "idbPOS2".f[18].p.read.mc.STATE;
    L "dbCONST".BLK.POS2.STATE.OPENED;
    ==I;
    );
    = #tIL.Source[1];

NETWORK
TITLE = Item 51 DV2113 interlock source : A RD2101 Vessel Burst Disc ALARM
    //------------------------------------------------------------------------//
    // Calculate the interlock condition:                                     //
    //------------------------------------------------------------------------//
    A idbDI1.f[14].p.read.mc.INTERLOCK;
    = #tIL.Source[2];

NETWORK
TITLE = Item 51 DV2113 interlock source : A ES2100 Vessel Emergency Stop mounted on HMI INTERLOCK
    //------------------------------------------------------------------------//
    // Calculate the interlock condition:                                     //
    //------------------------------------------------------------------------//
    A idbDI1.f[8].p.read.mc.INTERLOCK;
    = #tIL.Source[3];

NETWORK
TITLE = Item 51 DV2113 interlock source : A PI2103 Vessel Pressure Indicator INTERLOCK
    //------------------------------------------------------------------------//
    // Calculate the interlock condition:                                     //
    //------------------------------------------------------------------------//
    A idbPI1.f[1].p.read.mc.INTERLOCK;
    = #tIL.Source[4];

NETWORK
TITLE = Item 51 DV2113 interlock source : A ASL2000 Vessel Instrument Air Switch INTERLOCK
    //------------------------------------------------------------------------//
    // Calculate the interlock condition:                                     //
    //------------------------------------------------------------------------//
    A idbDI1.f[1].p.read.mc.INTERLOCK;
    = #tIL.Source[5];

NETWORK
TITLE = Item 51 DV2113 interlock source : AN ZSC2101 Vessel Manway Closed Indicator CLOSED
    //------------------------------------------------------------------------//
    // Calculate the interlock condition:                                     //
    //------------------------------------------------------------------------//
    AN(;
    L "idbZSC1".f[1].p.read.mc.STATE;
    L "dbCONST".BLK.ZSC1.STATE.CLOSED;
    ==I;
    );
    = #tIL.Source[6];

NETWORK
TITLE = Item 51 DV2113 interlock source : O MI2101 Mx Mass Indicator High High Alarm ALARM_HH   ON MI2101 Mx Mass Indicator Bad DQ DQ
    //------------------------------------------------------------------------//
    // Calculate the interlock condition:                                     //
    //------------------------------------------------------------------------//
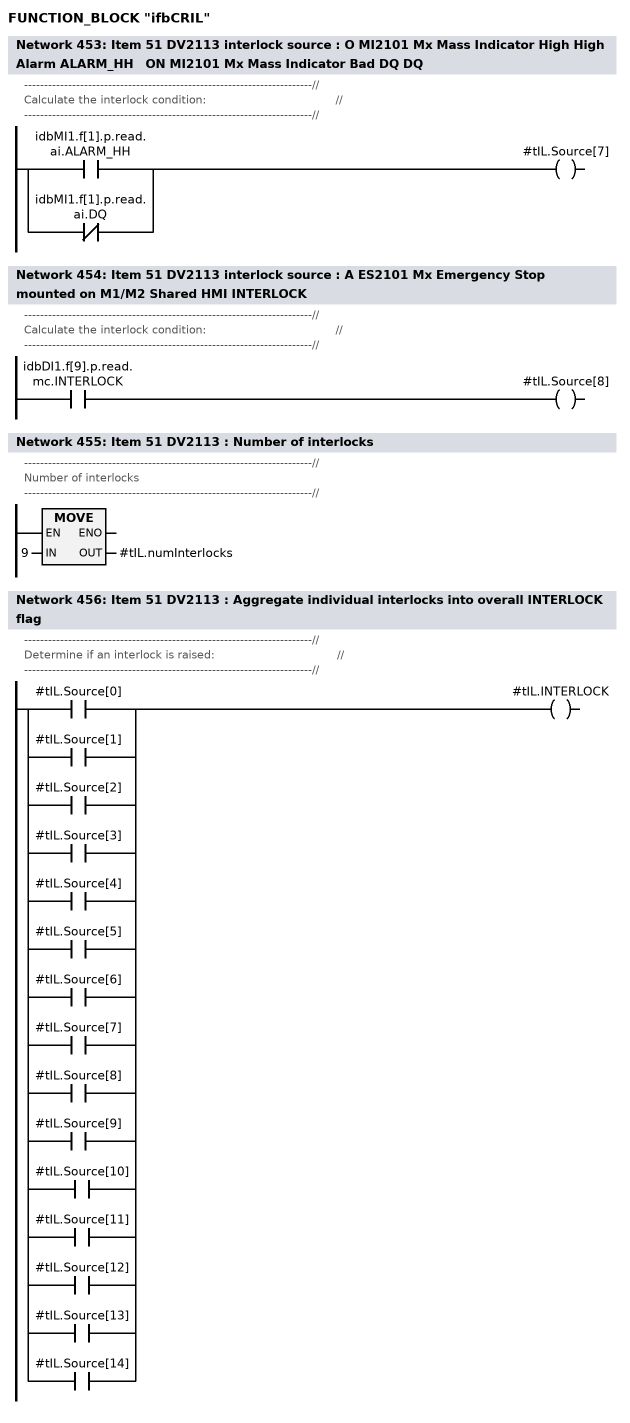
    O idbMI1.f[1].p.read.ai.ALARM_HH;
ON idbMI1.f[1].p.read.ai.DQ;
    = #tIL.Source[7];

NETWORK
TITLE = Item 51 DV2113 interlock source : A ES2101 Mx Emergency Stop mounted on M1/M2 Shared HMI INTERLOCK
    //------------------------------------------------------------------------//
    // Calculate the interlock condition:                                     //
    //------------------------------------------------------------------------//
    A idbDI1.f[9].p.read.mc.INTERLOCK;
    = #tIL.Source[8];


NETWORK
TITLE = Item 51 DV2113 : Number of interlocks
    //------------------------------------------------------------------------//
    // Number of interlocks
    //------------------------------------------------------------------------//
    L 9;
    T #tIL.numInterlocks;

NETWORK
TITLE = Item 51 DV2113 : Aggregate individual interlocks into overall INTERLOCK flag
    //------------------------------------------------------------------------//
    // Determine if an interlock is raised:                                   //
    //------------------------------------------------------------------------//
    O #tIL.Source[0];
    O #tIL.Source[1];
    O #tIL.Source[2];
    O #tIL.Source[3];
    O #tIL.Source[4];
    O #tIL.Source[5];
    O #tIL.Source[6];
    O #tIL.Source[7];
    O #tIL.Source[8];
    O #tIL.Source[9];
    O #tIL.Source[10];
    O #tIL.Source[11];
    O #tIL.Source[12];
    O #tIL.Source[13];
    O #tIL.Source[14];
    = #tIL.INTERLOCK;

NETWORK
TITLE = Item 51 DV2113 : Update the instance data
    //------------------------------------------------------------------------//
    // Update the instance DB with the calculated interlock flags:            //
    //------------------------------------------------------------------------//
    CALL MOVE
    {value_type := 'Variant'}
    (   IN                   := #tIL ,
        OUT                  := #p[51]
    );

NETWORK
TITLE = Item 52 DV2115 : PS Supply for PW Loop initialise variables
    //------------------------------------------------------------------------//
    // CRITICAL INTERLOCK   CRITICAL INTERLOCK   CRITICAL INTERLOCK   CRITICA //
    // CRITICAL INTERLOCK   CRITICAL INTERLOCK   CRITICAL INTERLOCK   CRITICA //
    //                                                                        //
    // Clear the interlock flag:                                              //
    //------------------------------------------------------------------------//
    A "alwaysLow";
    = #tIL.INTERLOCK;

    //------------------------------------------------------------------------//
    // Clear all interlock values to initialise them to off:                  //
    //------------------------------------------------------------------------//
    CALL FILL_BLK
    {value_type := 'Bool', count_type := 'UInt'}
    (   IN                   := 0 ,
        COUNT                := 15 ,
        OUT                  := #tIL.Source[0]
    );


NETWORK
TITLE = Item 52 DV2115 interlock source : ON ZSC2107 Vessel inlet line Flowpath Indicator IN   ON ZSC2105 Vessel PW Supply Flowpath Indicator IN
    //------------------------------------------------------------------------//
    // Calculate the interlock condition:                                     //
    //------------------------------------------------------------------------//
    ON(;
    L "idbZSC2".f[9].p.read.mc.STATE;
    L "dbCONST".BLK.ZSC2.STATE.IN;
    ==I;
    );
ON(;
    L "idbZSC2".f[8].p.read.mc.STATE;
    L "dbCONST".BLK.ZSC2.STATE.IN;
    ==I;
    );
    = #tIL.Source[0];

NETWORK
TITLE = Item 52 DV2115 interlock source : A DV2113 Vessel PW Supply Valve OPENED
    //------------------------------------------------------------------------//
    // Calculate the interlock condition:                                     //
    //------------------------------------------------------------------------//
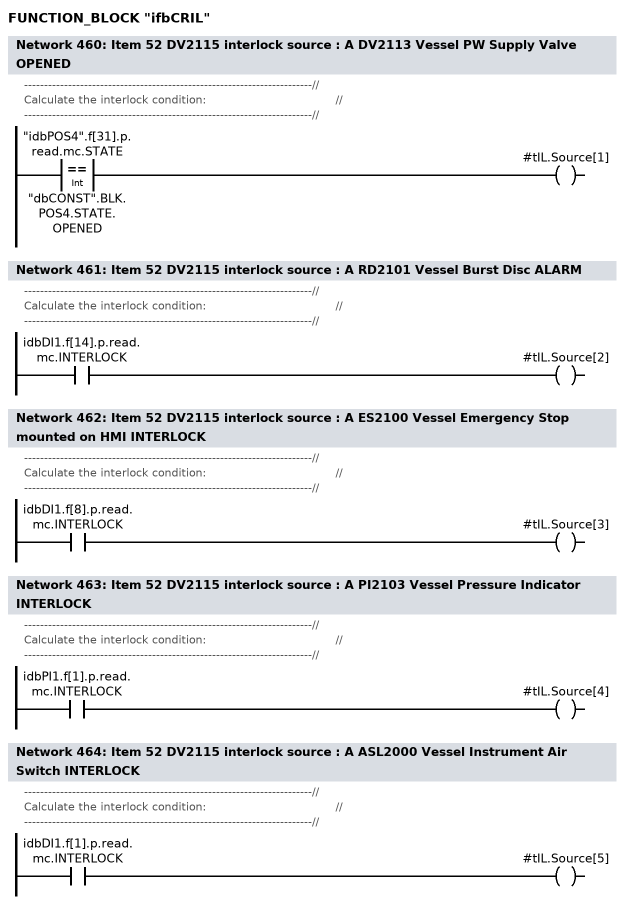
    A(;
    L "idbPOS4".f[31].p.read.mc.STATE;
    L "dbCONST".BLK.POS4.STATE.OPENED;
    ==I;
    );
    = #tIL.Source[1];

NETWORK
TITLE = Item 52 DV2115 interlock source : A RD2101 Vessel Burst Disc ALARM
    //------------------------------------------------------------------------//
    // Calculate the interlock condition:                                     //
    //------------------------------------------------------------------------//
    A idbDI1.f[14].p.read.mc.INTERLOCK;
    = #tIL.Source[2];

NETWORK
TITLE = Item 52 DV2115 interlock source : A ES2100 Vessel Emergency Stop mounted on HMI INTERLOCK
    //------------------------------------------------------------------------//
    // Calculate the interlock condition:                                     //
    //------------------------------------------------------------------------//
    A idbDI1.f[8].p.read.mc.INTERLOCK;
    = #tIL.Source[3];

NETWORK
TITLE = Item 52 DV2115 interlock source : A PI2103 Vessel Pressure Indicator INTERLOCK
    //------------------------------------------------------------------------//
    // Calculate the interlock condition:                                     //
    //------------------------------------------------------------------------//
    A idbPI1.f[1].p.read.mc.INTERLOCK;
    = #tIL.Source[4];

NETWORK
TITLE = Item 52 DV2115 interlock source : A ASL2000 Vessel Instrument Air Switch INTERLOCK
    //------------------------------------------------------------------------//
    // Calculate the interlock condition:                                     //
    //------------------------------------------------------------------------//
    A idbDI1.f[1].p.read.mc.INTERLOCK;
    = #tIL.Source[5];

NETWORK
TITLE = Item 52 DV2115 interlock source : AN ZSC2101 Vessel Manway Closed Indicator CLOSED
    //------------------------------------------------------------------------//
    // Calculate the interlock condition:                                     //
    //------------------------------------------------------------------------//
    AN(;
    L "idbZSC1".f[1].p.read.mc.STATE;
    L "dbCONST".BLK.ZSC1.STATE.CLOSED;
    ==I;
    );
    = #tIL.Source[6];

NETWORK
TITLE = Item 52 DV2115 interlock source : O MI2101 Mx Mass Indicator High High Alarm ALARM_HH   ON MI2101 Mx Mass Indicator Bad DQ DQ
    //------------------------------------------------------------------------//
    // Calculate the interlock condition:                                     //
    //------------------------------------------------------------------------//
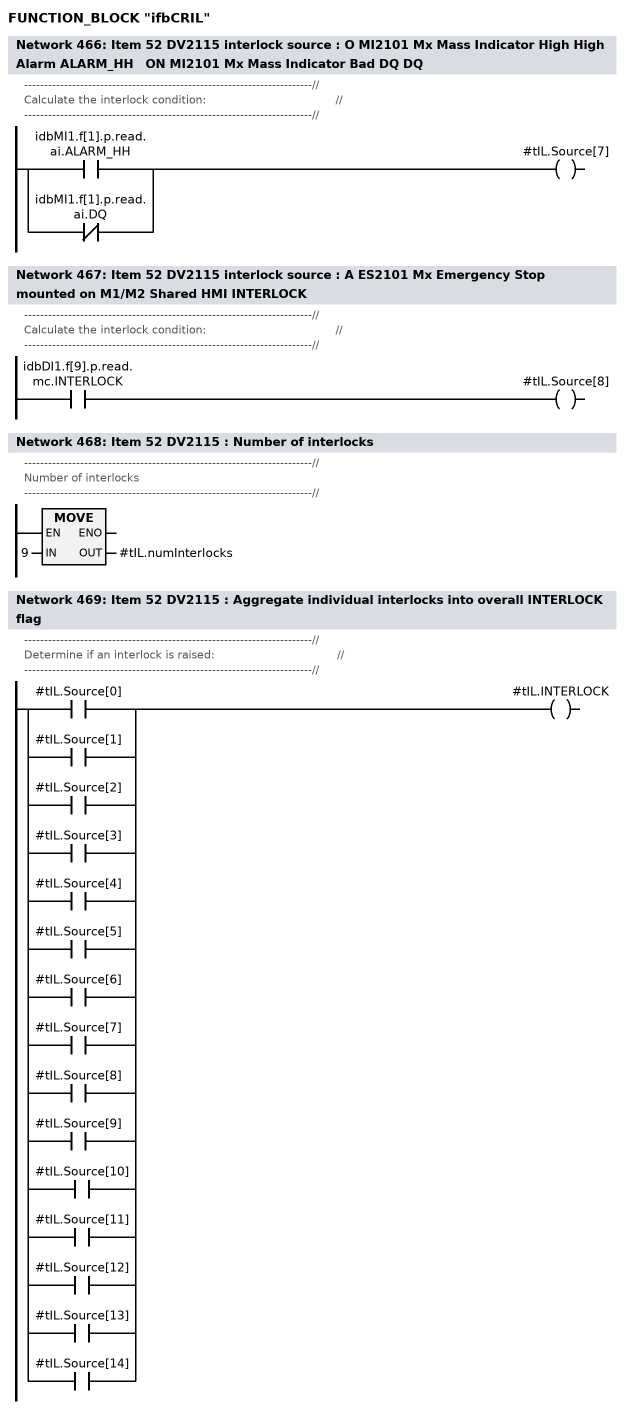
    O idbMI1.f[1].p.read.ai.ALARM_HH;
ON idbMI1.f[1].p.read.ai.DQ;
    = #tIL.Source[7];

NETWORK
TITLE = Item 52 DV2115 interlock source : A ES2101 Mx Emergency Stop mounted on M1/M2 Shared HMI INTERLOCK
    //------------------------------------------------------------------------//
    // Calculate the interlock condition:                                     //
    //------------------------------------------------------------------------//
    A idbDI1.f[9].p.read.mc.INTERLOCK;
    = #tIL.Source[8];


NETWORK
TITLE = Item 52 DV2115 : Number of interlocks
    //------------------------------------------------------------------------//
    // Number of interlocks
    //------------------------------------------------------------------------//
    L 9;
    T #tIL.numInterlocks;

NETWORK
TITLE = Item 52 DV2115 : Aggregate individual interlocks into overall INTERLOCK flag
    //------------------------------------------------------------------------//
    // Determine if an interlock is raised:                                   //
    //------------------------------------------------------------------------//
    O #tIL.Source[0];
    O #tIL.Source[1];
    O #tIL.Source[2];
    O #tIL.Source[3];
    O #tIL.Source[4];
    O #tIL.Source[5];
    O #tIL.Source[6];
    O #tIL.Source[7];
    O #tIL.Source[8];
    O #tIL.Source[9];
    O #tIL.Source[10];
    O #tIL.Source[11];
    O #tIL.Source[12];
    O #tIL.Source[13];
    O #tIL.Source[14];
    = #tIL.INTERLOCK;

NETWORK
TITLE = Item 52 DV2115 : Update the instance data
    //------------------------------------------------------------------------//
    // Update the instance DB with the calculated interlock flags:            //
    //------------------------------------------------------------------------//
    CALL MOVE
    {value_type := 'Variant'}
    (   IN                   := #tIL ,
        OUT                  := #p[52]
    );

NETWORK
TITLE = Item 53 DV2117 : Spray Ball 1 Valve initialise variables
    //------------------------------------------------------------------------//
    // CRITICAL INTERLOCK   CRITICAL INTERLOCK   CRITICAL INTERLOCK   CRITICA //
    // CRITICAL INTERLOCK   CRITICAL INTERLOCK   CRITICAL INTERLOCK   CRITICA //
    //                                                                        //
    // Clear the interlock flag:                                              //
    //------------------------------------------------------------------------//
    A "alwaysLow";
    = #tIL.INTERLOCK;

    //------------------------------------------------------------------------//
    // Clear all interlock values to initialise them to off:                  //
    //------------------------------------------------------------------------//
    CALL FILL_BLK
    {value_type := 'Bool', count_type := 'UInt'}
    (   IN                   := 0 ,
        COUNT                := 15 ,
        OUT                  := #tIL.Source[0]
    );


NETWORK
TITLE = Item 53 DV2117 interlock source : A RD2101 Vessel Burst Disc ALARM
    //------------------------------------------------------------------------//
    // Calculate the interlock condition:                                     //
    //------------------------------------------------------------------------//
    A idbDI1.f[14].p.read.mc.INTERLOCK;
    = #tIL.Source[0];

NETWORK
TITLE = Item 53 DV2117 interlock source : A ES2100 Vessel Emergency Stop mounted on HMI INTERLOCK
    //------------------------------------------------------------------------//
    // Calculate the interlock condition:                                     //
    //------------------------------------------------------------------------//
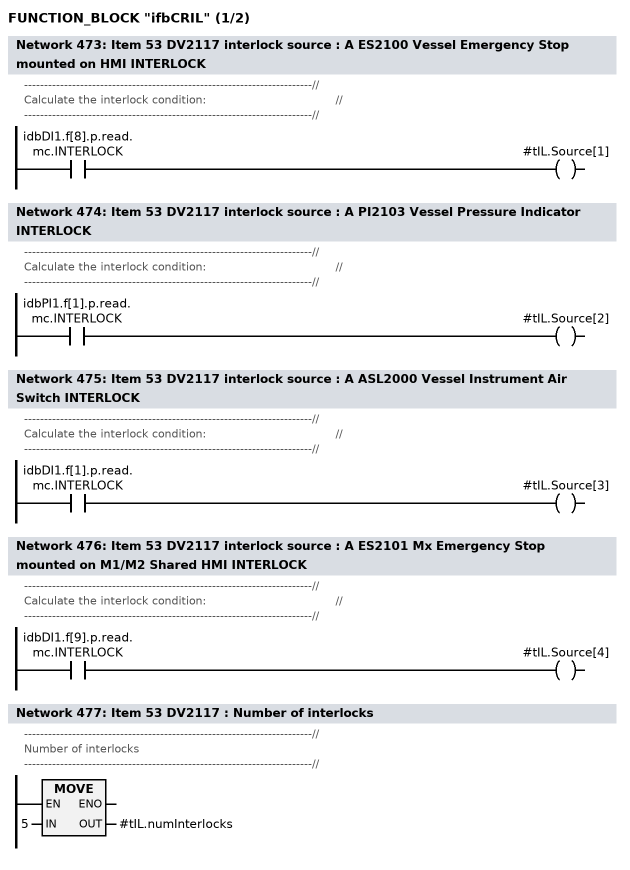
    A idbDI1.f[8].p.read.mc.INTERLOCK;
    = #tIL.Source[1];

NETWORK
TITLE = Item 53 DV2117 interlock source : A PI2103 Vessel Pressure Indicator INTERLOCK
    //------------------------------------------------------------------------//
    // Calculate the interlock condition:                                     //
    //------------------------------------------------------------------------//
    A idbPI1.f[1].p.read.mc.INTERLOCK;
    = #tIL.Source[2];

NETWORK
TITLE = Item 53 DV2117 interlock source : A ASL2000 Vessel Instrument Air Switch INTERLOCK
    //------------------------------------------------------------------------//
    // Calculate the interlock condition:                                     //
    //------------------------------------------------------------------------//
    A idbDI1.f[1].p.read.mc.INTERLOCK;
    = #tIL.Source[3];

NETWORK
TITLE = Item 53 DV2117 interlock source : A ES2101 Mx Emergency Stop mounted on M1/M2 Shared HMI INTERLOCK
    //------------------------------------------------------------------------//
    // Calculate the interlock condition:                                     //
    //------------------------------------------------------------------------//
    A idbDI1.f[9].p.read.mc.INTERLOCK;
    = #tIL.Source[4];


NETWORK
TITLE = Item 53 DV2117 : Number of interlocks
    //------------------------------------------------------------------------//
    // Number of interlocks
    //------------------------------------------------------------------------//
    L 5;
    T #tIL.numInterlocks;

NETWORK
TITLE = Item 53 DV2117 : Aggregate individual interlocks into overall INTERLOCK flag
    //------------------------------------------------------------------------//
    // Determine if an interlock is raised:                                   //
    //------------------------------------------------------------------------//
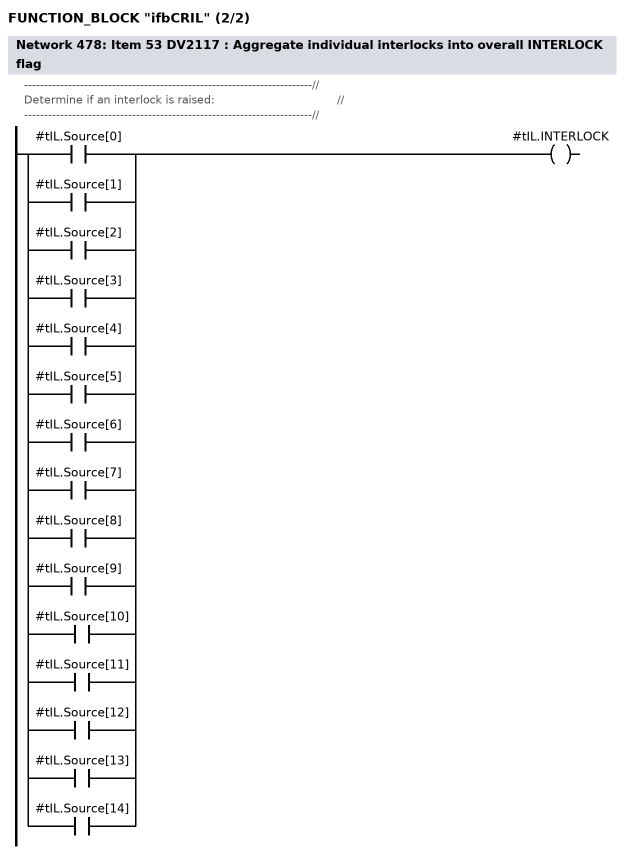
    O #tIL.Source[0];
    O #tIL.Source[1];
    O #tIL.Source[2];
    O #tIL.Source[3];
    O #tIL.Source[4];
    O #tIL.Source[5];
    O #tIL.Source[6];
    O #tIL.Source[7];
    O #tIL.Source[8];
    O #tIL.Source[9];
    O #tIL.Source[10];
    O #tIL.Source[11];
    O #tIL.Source[12];
    O #tIL.Source[13];
    O #tIL.Source[14];
    = #tIL.INTERLOCK;

NETWORK
TITLE = Item 53 DV2117 : Update the instance data
    //------------------------------------------------------------------------//
    // Update the instance DB with the calculated interlock flags:            //
    //------------------------------------------------------------------------//
    CALL MOVE
    {value_type := 'Variant'}
    (   IN                   := #tIL ,
        OUT                  := #p[53]
    );

NETWORK
TITLE = Item 54 DV2119 : Spray Ball 2 Valve initialise variables
    //------------------------------------------------------------------------//
    // CRITICAL INTERLOCK   CRITICAL INTERLOCK   CRITICAL INTERLOCK   CRITICA //
    // CRITICAL INTERLOCK   CRITICAL INTERLOCK   CRITICAL INTERLOCK   CRITICA //
    //                                                                        //
    // Clear the interlock flag:                                              //
    //------------------------------------------------------------------------//
    A "alwaysLow";
    = #tIL.INTERLOCK;

    //------------------------------------------------------------------------//
    // Clear all interlock values to initialise them to off:                  //
    //------------------------------------------------------------------------//
    CALL FILL_BLK
    {value_type := 'Bool', count_type := 'UInt'}
    (   IN                   := 0 ,
        COUNT                := 15 ,
        OUT                  := #tIL.Source[0]
    );


NETWORK
TITLE = Item 54 DV2119 interlock source : A RD2101 Vessel Burst Disc ALARM
    //------------------------------------------------------------------------//
    // Calculate the interlock condition:                                     //
    //------------------------------------------------------------------------//
    A idbDI1.f[14].p.read.mc.INTERLOCK;
    = #tIL.Source[0];

NETWORK
TITLE = Item 54 DV2119 interlock source : A ES2100 Vessel Emergency Stop mounted on HMI INTERLOCK
    //------------------------------------------------------------------------//
    // Calculate the interlock condition:                                     //
    //------------------------------------------------------------------------//
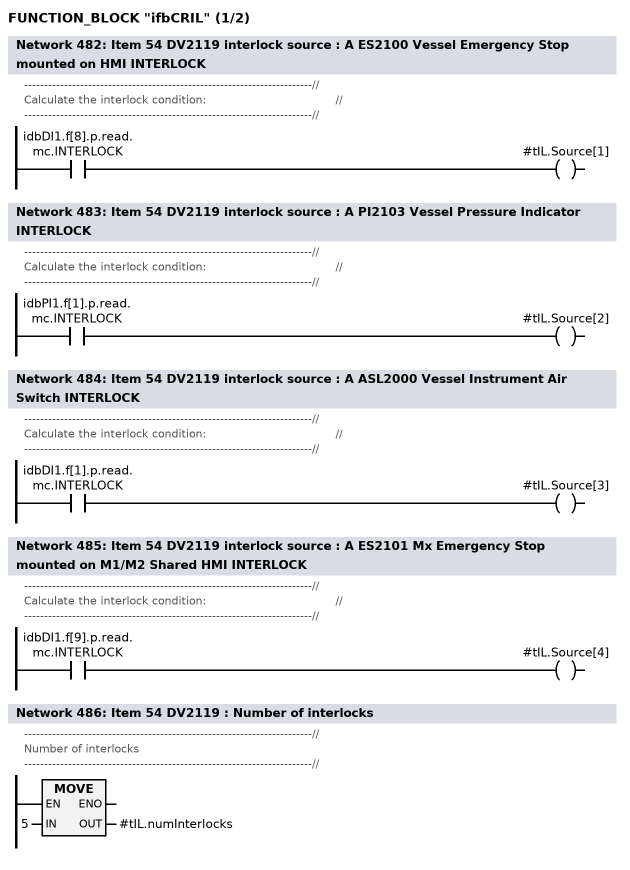
    A idbDI1.f[8].p.read.mc.INTERLOCK;
    = #tIL.Source[1];

NETWORK
TITLE = Item 54 DV2119 interlock source : A PI2103 Vessel Pressure Indicator INTERLOCK
    //------------------------------------------------------------------------//
    // Calculate the interlock condition:                                     //
    //------------------------------------------------------------------------//
    A idbPI1.f[1].p.read.mc.INTERLOCK;
    = #tIL.Source[2];

NETWORK
TITLE = Item 54 DV2119 interlock source : A ASL2000 Vessel Instrument Air Switch INTERLOCK
    //------------------------------------------------------------------------//
    // Calculate the interlock condition:                                     //
    //------------------------------------------------------------------------//
    A idbDI1.f[1].p.read.mc.INTERLOCK;
    = #tIL.Source[3];

NETWORK
TITLE = Item 54 DV2119 interlock source : A ES2101 Mx Emergency Stop mounted on M1/M2 Shared HMI INTERLOCK
    //------------------------------------------------------------------------//
    // Calculate the interlock condition:                                     //
    //------------------------------------------------------------------------//
    A idbDI1.f[9].p.read.mc.INTERLOCK;
    = #tIL.Source[4];


NETWORK
TITLE = Item 54 DV2119 : Number of interlocks
    //------------------------------------------------------------------------//
    // Number of interlocks
    //------------------------------------------------------------------------//
    L 5;
    T #tIL.numInterlocks;

NETWORK
TITLE = Item 54 DV2119 : Aggregate individual interlocks into overall INTERLOCK flag
    //------------------------------------------------------------------------//
    // Determine if an interlock is raised:                                   //
    //------------------------------------------------------------------------//
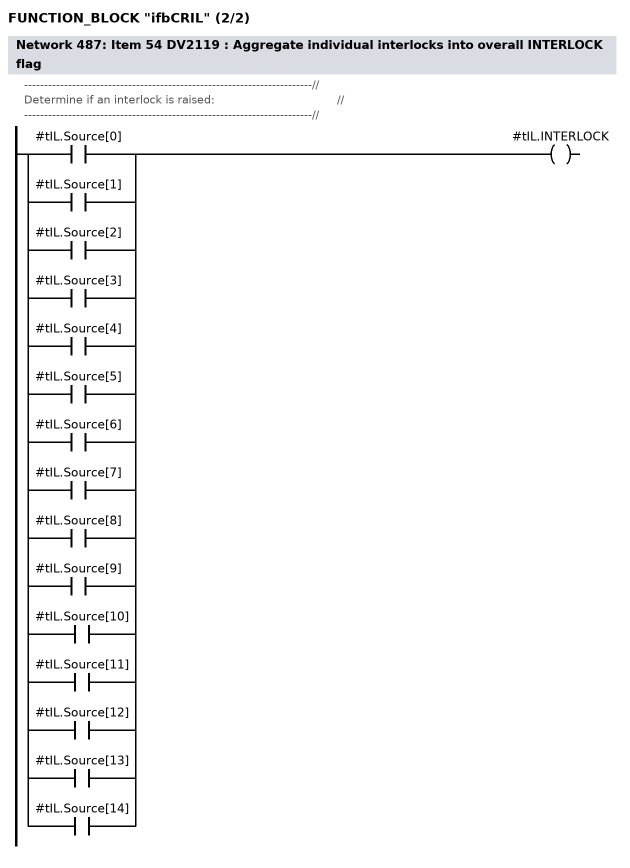
    O #tIL.Source[0];
    O #tIL.Source[1];
    O #tIL.Source[2];
    O #tIL.Source[3];
    O #tIL.Source[4];
    O #tIL.Source[5];
    O #tIL.Source[6];
    O #tIL.Source[7];
    O #tIL.Source[8];
    O #tIL.Source[9];
    O #tIL.Source[10];
    O #tIL.Source[11];
    O #tIL.Source[12];
    O #tIL.Source[13];
    O #tIL.Source[14];
    = #tIL.INTERLOCK;

NETWORK
TITLE = Item 54 DV2119 : Update the instance data
    //------------------------------------------------------------------------//
    // Update the instance DB with the calculated interlock flags:            //
    //------------------------------------------------------------------------//
    CALL MOVE
    {value_type := 'Variant'}
    (   IN                   := #tIL ,
        OUT                  := #p[54]
    );

NETWORK
TITLE = Item 55 DV2121 : Outlet Valve initialise variables
    //------------------------------------------------------------------------//
    // CRITICAL INTERLOCK   CRITICAL INTERLOCK   CRITICAL INTERLOCK   CRITICA //
    // CRITICAL INTERLOCK   CRITICAL INTERLOCK   CRITICAL INTERLOCK   CRITICA //
    //                                                                        //
    // Clear the interlock flag:                                              //
    //------------------------------------------------------------------------//
    A "alwaysLow";
    = #tIL.INTERLOCK;

    //------------------------------------------------------------------------//
    // Clear all interlock values to initialise them to off:                  //
    //------------------------------------------------------------------------//
    CALL FILL_BLK
    {value_type := 'Bool', count_type := 'UInt'}
    (   IN                   := 0 ,
        COUNT                := 15 ,
        OUT                  := #tIL.Source[0]
    );


NETWORK
TITLE = Item 55 DV2121 interlock source : A RD2101 Vessel Burst Disc ALARM
    //------------------------------------------------------------------------//
    // Calculate the interlock condition:                                     //
    //------------------------------------------------------------------------//
    A idbDI1.f[14].p.read.mc.INTERLOCK;
    = #tIL.Source[0];

NETWORK
TITLE = Item 55 DV2121 interlock source : A ES2100 Vessel Emergency Stop mounted on HMI INTERLOCK
    //------------------------------------------------------------------------//
    // Calculate the interlock condition:                                     //
    //------------------------------------------------------------------------//
